{attribute 'obsolete' := 'No longer any reason to use this, all state classes can have unit tests.'}
FUNCTION_BLOCK FB_PositionStatePMPS_Test EXTENDS FB_PositionStatePMPS_Base
(*
    Implement position state pmps with no FFO and auto-accept transition after 3s
    Use for offline testing of everything except the explicit interface
*)
VAR
    tonReq: TON;
END_VAR


Exec();

ACTION HandleBPTM:

// Send the fake BPTM our assertion request by changing stStateReq.stBeamParams
// We expect to recieve bTransitionAuthorized TRUE after some delta T
// We expect bTransitionAuthorized to go FALSE after stMotionStage.bBusy goes FALSE
tonReq(
    IN:=bInTransition,
    PT:=T#3s);
bTransitionAuthorized := tonReq.Q AND stMotionStage.bExecute;
END_ACTION

ACTION HandleFFO:

// Skip implementing this for offline testing
// We won't be able to tell if it worked anyway
END_ACTION

END_FUNCTION_BLOCK

(* stored: Version 1.1.0.1
   POU FB_PositionStatePMPS_Test: Id {116f57d8-27d2-44f6-a73e-8c9b24b1bd3d}, SpecialFunc None
   Action HandleBPTM: Id {a1c65ced-35d8-47df-ada1-08298070502e}
   Action HandleFFO: Id {bbf94cf3-04b5-4757-809d-723da17dcc32} *)
